// TIA Portal V18 export
VAR_GLOBAL   // PLC tag table "Tabella delle variabili standard"
END_VAR
